Fanuc KAREL source: kb00035.KL

PROGRAM KB00035
%NOLOCKGROUP
VAR
P1:INTEGER;P2:INTEGER;P3:INTEGER;P4 : STRING[80]
BEGIN
--
--
--
P1=1
P2=1
P3=1
P4='A'
CNV_INT_STR(P1,P2,P3,P4)
END KB00035
